FUNCTION_BLOCK FB_Child1 EXTENDS FB_Parent
VAR
	
END_VAR

METHOD  Eat
VAR_INPUT
END_VAR
sOutput:= 'Child is eating ';
END_METHOD

METHOD  Greet 
VAR_INPUT
END_VAR
sOutput:= 'Child is greeting';
END_METHOD

END_FUNCTION_BLOCK

(* stored: Version 1.1.0.1, ProductVersion 3.1.4024.16
   POU FB_Child1: Id {fc5ffea7-5e51-4d8e-b3a4-23013a0a7b75}, SpecialFunc None
   Method Eat: Id {eeef6ae9-f238-4ae6-931b-1d18f91c0086}
   Method Greet: Id {10690703-0695-4f79-b32e-8ed40438a1d4} *)
